PROGRAM MAIN
VAR

END_VAR


PRG_ZF_Control();
PRG_Engine();
PRG_BlinkMarine();
PRG_Ballast();
PRG_Doors();
PRG_Winches();
PRG_SimDoors();
PRG_HmiLeds();

END_PROGRAM

(* stored: Version 1.1.0.1, ProductVersion 3.1.4026.17
   POU MAIN: Id {7b9c8698-7ce0-48af-9cd6-368a0771761d}, SpecialFunc None *)
